(* CODESYS project Mbc_Tc3_Pcs_v1.0.0.1.library
   Company: mbc engineering GmbH
   DefaultNamespace: Mbc_Tc3_Pcs
   Version: 1.0.0.1
   Placeholder: MBC TC3 PCS Library
   Author: mbc engineering GmbH
   DocFormat: reStructuredText
   Title: MBC TC3 PCS Library

Project tree, tasks and I/O mapping:
  Command/
    function block CommandBase [ST]: Abort, CalculateProgress, Done, Refresh, Task
    data type E_CommandResultCode
    interface ICommand: Refresh
    data type ST_CommandBaseHandshake
  docs/
    Readme.md
  Version/
    global variables Global_Version
  Mbc_Tc3_Pcs.tmc
*)

// Command/E_CommandResultCode
{attribute 'qualified_only'}
{attribute 'strict'}
TYPE E_CommandResultCode :
(
	Init := 0,
	Running := 1,
	Done := 2,
	Cancelled := 3
) UINT;
END_TYPE

// Command/ST_CommandBaseHandshake
TYPE ST_CommandBaseHandshake :
STRUCT
	bExecute		: BOOL;		// Will be set to true from the PCS to start the command. When the operation are finish, the PLC will set the to false. On a long running Task, the PCS can reset to false for Abort the operation. 
	bBusy			: BOOL;		// When the operation is running. Only for multible cycle operations.
	nResultCode		: UINT;		// Shows the operation result code of the commando state. Default Values see 'CommandResultCode' Enum Type.
	nProgress		: UINT;		// Shows the optional calculated progress. The value is depend on the button implementation. (default can be 0..100%). Only necessary on long running operations.
END_STRUCT
END_TYPE

// Version/Global_Version
{attribute 'TcGenerated'}
// This function has been automatically generated from the project information.
VAR_GLOBAL CONSTANT
	{attribute 'const_non_replaced'}
	{attribute 'linkalways'}
	stLibVersion_MBC_TC3_PCS_Library : ST_LibVersion := (iMajor := 1, iMinor := 0, iBuild := 0, iRevision := 1, sVersion := '1.0.0.1');
END_VAR

// Command/CommandBase
FUNCTION_BLOCK PUBLIC CommandBase IMPLEMENTS ICommand
VAR_IN_OUT
	(* Use Class Properties for IN_OUT Parameters!!! *)
END_VAR
VAR PERSISTENT
	stHandshake		: ST_CommandBaseHandshake;		// Variable Strukture for communication with PCS. Aditional IN and OUT parameters should be declared in the derived implementation.
END_VAR

// OO-Class 
;

// Stops execution of Command 
METHOD PUBLIC Abort
stHandshake.nResultCode := E_CommandResultCode.Cancelled;
stHandshake.bExecute := FALSE;
stHandshake.bBusy := FALSE;
END_METHOD

METHOD PROTECTED CalculateProgress
IF stHandshake.nResultCode = E_CommandResultCode.Done THEN
	stHandshake.nProgress := 100;
ELSE
	stHandshake.nProgress := 0;
END_IF
END_METHOD

METHOD PROTECTED Done
stHandshake.nResultCode := E_CommandResultCode.Done;
stHandshake.bExecute := FALSE;
stHandshake.bBusy := FALSE;
END_METHOD

// Update the state of the command button. Should be called every cycle.
METHOD PUBLIC Refresh
VAR
	bInit		: BOOL;
END_VAR
// Starting Case
stHandshake.bBusy S= bInit := stHandshake.bExecute AND NOT stHandshake.bBusy;

// Reset Case
IF NOT stHandshake.bExecute AND stHandshake.bBusy THEN
	Abort();
END_IF

// Running Case
IF stHandshake.bExecute AND stHandshake.bBusy THEN
	IF bInit THEN
		stHandshake.nResultCode := E_CommandResultCode.Running;
	END_IF
	
	// Set Task init on First Call
	IF Task(bInit) THEN
		Done();
	END_IF
	
	CalculateProgress();
END_IF
END_METHOD

// Execute the funktional part of the command implementation
METHOD PROTECTED Task : BOOL
VAR_INPUT
	Init 	: BOOL;		// True the first time the Task is called after Execute is started
END_VAR
// Task complete if return true
Task := TRUE;
END_METHOD

END_FUNCTION_BLOCK

// Command/ICommand
INTERFACE ICommand

METHOD Refresh
END_METHOD

END_INTERFACE
